ABB RAPID module: RobData.sys

%%%
  VERSION:1
  LANGUAGE:ENGLISH
%%%

MODULE RobData(SYSMODULE)
  PERS tooldata tMaster:=[TRUE,[[-89.5851,55.1764,553.649],[1,0,0,0]],[175,[210,0,310],[1,0,0,0],15,15,15]];
  LOCAL CONST string stModuleName:="robdata";
  !
  ! Mission Routine Names
  !------------------------------------
  !
  CONST string stMissionNames{12}:=["PrelCarro1","PrelCarro2","DepCNC","PrelCNC","DepCarro1","DepCarro2","DepOut","DepIsp","PrelIsp","DepMeasure","PrelMeasure","Scarto"];
  !
  !ToolData
  PERS tooldata tPinzaA:=[TRUE,[[-361.2,0,367],[0.5,-0.5,-0.5,0.5]],[47.9,[0.7,0,403.9],[1,0,0,0],0,0,1.813]];
  PERS tooldata tPinzaB:=[TRUE,[[361.2,0,367],[0.5,0.5,0.5,0.5]],[47.9,[0.7,0,403.9],[1,0,0,0],0,0,0]];
  !WobjData
  !PERS wobjdata wRowSX:=[FALSE,TRUE,"",[[1120.43,789.859,397.66],[0.701994,0.001537,-0.00145,0.712186]],[[0,0,0],[1,0,0,0]]];
  PERS wobjdata wRowSX:=[FALSE,TRUE,"",[[1120.43,789.859,397.66],[0.701996,-0.000301,0.000415,0.712187]],[[0,0,0],[1,0,0,0]]];
  PERS wobjdata wRowDX:=[FALSE,TRUE,"",[[1091.49,-748.057,393.703],[0.00356,0.709853,-0.704334,0.003074]],[[-0.006557,0.001788,-0.001043],[1,0,0,-1E-06]]];
  !   Posizioni di servizio Fuori Ingombrom (FI)
  CONST jointtarget jFI_OffLine:=[[0,-20,-40,0,60,0],[9E+09,9E+09,9E+09,9E+09,9E+09,9E+09]];
  CONST jointtarget jFI_Manut:=[[31.22,16.05,8.21,-0.01,65.91,86.62],[9E+09,9E+09,9E+09,9E+09,9E+09,9E+09]];
  !CONST jointtarget jHomePos:=[[0,-45,15,0,30,90],[9E+09,9E+09,9E+09,9E+09,9E+09,9E+09]];
  CONST jointtarget jHomePos:=[[-7.29,-46.66,20.73,0,108.69,84.36],[9E+09,9E+09,9E+09,9E+09,9E+09,9E+09]];
  CONST jointtarget jApp_A:=[[66.48,-5,22.73,62.95,104.66,65.03],[9E+09,9E+09,9E+09,9E+09,9E+09,9E+09]];
  CONST jointtarget jApp_B:=[[-74.1,-9.74,25.52,-61.45,97.11,-68.92],[9E+09,9E+09,9E+09,9E+09,9E+09,9E+09]];
  CONST jointtarget jFronteC2:=[[-90.41,-35.55,23.23,0,98.45,89.96],[9E+09,9E+09,9E+09,9E+09,9E+09,9E+09]];
  CONST jointtarget jFronteC1:=[[90.58,-35.64,23.49,0,98.28,89.96],[9E+09,9E+09,9E+09,9E+09,9E+09,9E+09]];
  CONST jointtarget jFronteOUT:=[[-45,-35.8,23.98,0,97.95,89.96],[9E+09,9E+09,9E+09,9E+09,9E+09,9E+09]];
  CONST jointtarget jFronteIsp:=[[-143.6,-35.65,23.52,0,98.26,89.96],[9E+09,9E+09,9E+09,9E+09,9E+09,9E+09]];
  CONST jointtarget jAppDepCNC:=[[70.95,-17.31,51.57,-31.31,-38.79,204.59],[9E+09,9E+09,9E+09,9E+09,9E+09,9E+09]];
  CONST jointtarget jAppPrelCNC:=[[70.95,-17.31,51.57,-31.31,-38.79,25.3],[9E+09,9E+09,9E+09,9E+09,9E+09,9E+09]];
  CONST jointtarget jApp_B_Dep:=[[-79.73,-14.71,16.17,-64.55,98.7,96.89],[9E+09,9E+09,9E+09,9E+09,9E+09,9E+09]];
  CONST jointtarget jApp_A_Dep:=[[79.94,-12.29,18.86,60.75,93.84,-100.21],[9E+09,9E+09,9E+09,9E+09,9E+09,9E+09]];
  CONST jointtarget jAppMeas:=[[-7.29,-46.66,27.39,0,108.69,84.36],[9E+09,9E+09,9E+09,9E+09,9E+09,9E+09]];
  CONST jointtarget jAppDepOut:=[[-56.48,9.2,9.11,101.75,58.38,-112.15],[9E+09,9E+09,9E+09,9E+09,9E+09,9E+09]];
  CONST jointtarget jOverBin:=[[-41.97,28.29,10.41,110.5,45.21,-131.89],[9E+09,9E+09,9E+09,9E+09,9E+09,9E+09]];
  CONST jointtarget jAppIsp:=[[-105,-5.17,33.52,-96.28,76.22,118.04],[9E+09,9E+09,9E+09,9E+09,9E+09,9E+09]];
  CONST jointtarget jSvincolo:=[[12.8571,-26.4171,21.7139,-68.3652,75.6916,118.136],[9E+09,9E+09,9E+09,9E+09,9E+09,9E+09]];
  CONST jointtarget jBackHome1:=[[90,-52.56,15.28,0,37.28,90],[9E+09,9E+09,9E+09,9E+09,9E+09,9E+09]];
  CONST jointtarget jBackHome2:=[[-90.15,-51.5,15.35,0.26,36.15,89.79],[9E+09,9E+09,9E+09,9E+09,9E+09,9E+09]];
  CONST robtarget pWayToDep:=[[1413.06,181.45,1150.37],[0.00963,-0.119155,0.989815,0.077305],[0,-1,1,0],[9E+09,9E+09,9E+09,9E+09,9E+09,9E+09]];
  CONST robtarget pWayToPrel:=[[1413.05,181.47,1150.32],[0.009594,-0.119153,0.989815,0.077319],[0,-1,1,0],[9E+09,9E+09,9E+09,9E+09,9E+09,9E+09]];

  !
ENDMODULE
